{attribute 'GeneratedUsingTerminal: EPP1111-0000-0016'}
{attribute addProperty BoxType "EPP1111-0000-0016"}
{attribute addProperty Id "ID_InputsAT %I*ID_Inputs_07C9D28F2WcStateAT %I*WcState_9091E0EB2InfoDataAT %I*InfoData_94A18F5E2"}
{attribute addProperty CRC "3053365944"}
{attribute addProperty Size "6"}
TYPE EPP1111_B5FEAAB8 EXTENDS EtcSlaveTerminalBase_947E5A46 :
STRUCT
	{attribute addProperty Name "ID_Inputs"}
	ID_Inputs : ID_Inputs_07C9D28F;
	{attribute addProperty Name "WcState"}
	WcState : WcState_9091E0EB;
	{attribute addProperty Name "InfoData"}
	InfoData : InfoData_94A18F5E;
END_STRUCT
END_TYPE

(* stored: Version 1.2.0.0, ProductVersion 3.1.4024.9
   DUT EPP1111_B5FEAAB8: Id {6f9e9022-b2be-4506-8b93-0c9d551ca27e} *)
